// TIA Portal V19 export
DATA_BLOCK "HmiInterface"   // DB39
// stored: Access Published, MemoryReserve 100, Namespace Unit2.EM4
   VAR
      em : "LAF_typeEmInterface";
      jobs : "LAF_typeJobsInterface";
      sequence : "LAF_typeSequenceInterface";
      cm1AxisControl { S7_SetPoint := 'True'} : "LBC_typeAxisSimpleControlInterface_1";
      cm2AxisControl { S7_SetPoint := 'True'} : "LBC_typeAxisSimpleControlInterface_1";
      cm3AxisControl { S7_SetPoint := 'True'} : "LBC_typeAxisSimpleControlInterface_1";
      cm4Cylinder { S7_SetPoint := 'True'} : "LBC_Simple_typeTwoWayActuatorInterface";
      cm5Cylinder { S7_SetPoint := 'True'} : "LBC_Simple_typeTwoWayActuatorInterface";
      cm6Cylinder { S7_SetPoint := 'True'} : "LBC_Simple_typeTwoWayActuatorInterface";
      cm7Cylinder { S7_SetPoint := 'True'} : "LBC_Simple_typeTwoWayActuatorInterface";
      cm8SignalTM { S7_SetPoint := 'True'} : "LEXCHANGETRAY_typeHandlingXyzIoSignalInterface";
      em4Parameters : "LAF_typeXyzhandlingEm4ParametersInterface";
   END_VAR
BEGIN
   // em4Parameters.configuration.cm1Axis119 : X
   // em4Parameters.configuration.cm2Axis120 : Y
   // em4Parameters.configuration.cm3Axis121 : Z
END_DATA_BLOCK
